FUNCTION_BLOCK Equipo_Valvula_5_2
VAR_INPUT
	PE 	  					  : BOOL;	//Parada de emergência
	Modo_Automatico           : BOOL;	//Modo automático
	Cmd_Auto         		  : BOOL;	//Comando automático
	Valv_Abierta		   	  : BOOL;	//Válvula aberta
	Valv_Cerrada			  : BOOL;	//Válvula fechada
	T_Discrepancia            : TIME;	//Tempo para erro de abertura
END_VAR
VAR_OUTPUT
	Activa_Equipo	 	      : BOOL;	//Aciona equipamento
	Estado					  : INT;	//Status da válvula
	Alr_Discrepancia		  : BOOL;	//Alarme de falha no acionamento
END_VAR
VAR_IN_OUT
	Cmd_Man 				  : BOOL;	//Comando manual
	Alarma				      : BOOL;	//Alarme
	Reset_Alarma		      : BOOL;	//Reset alarmes
END_VAR
VAR_STAT
	FP_Reset				  : R_TRIG;
	FN_Parada_Auto			  : F_TRIG;
	FP_Marcha_Auto            : R_TRIG;
	Cmd_Auto_interno		  :BOOL;	
END_VAR

VAR PERSISTENT
	Reset_Eventos         	  : BOOL;
	Timer_Discrepancia		  : TON;
	TON_TempoAbertura: TON;
	R_TRIG_TempoAbertura: R_TRIG;
	TempoAbertura	:DINT;	//Tempo que a válvula demora para abrir
	Eventos_Parciales		  : DINT;
	Eventos_Totales			  : DINT;
END_VAR
VAR // added by the converter: edge detectors and wires of the graphical bodies
    _w1, _w2, _w3, _w4, _w5, _w6, _w7 : BOOL;
    _rt1 : R_TRIG;
END_VAR

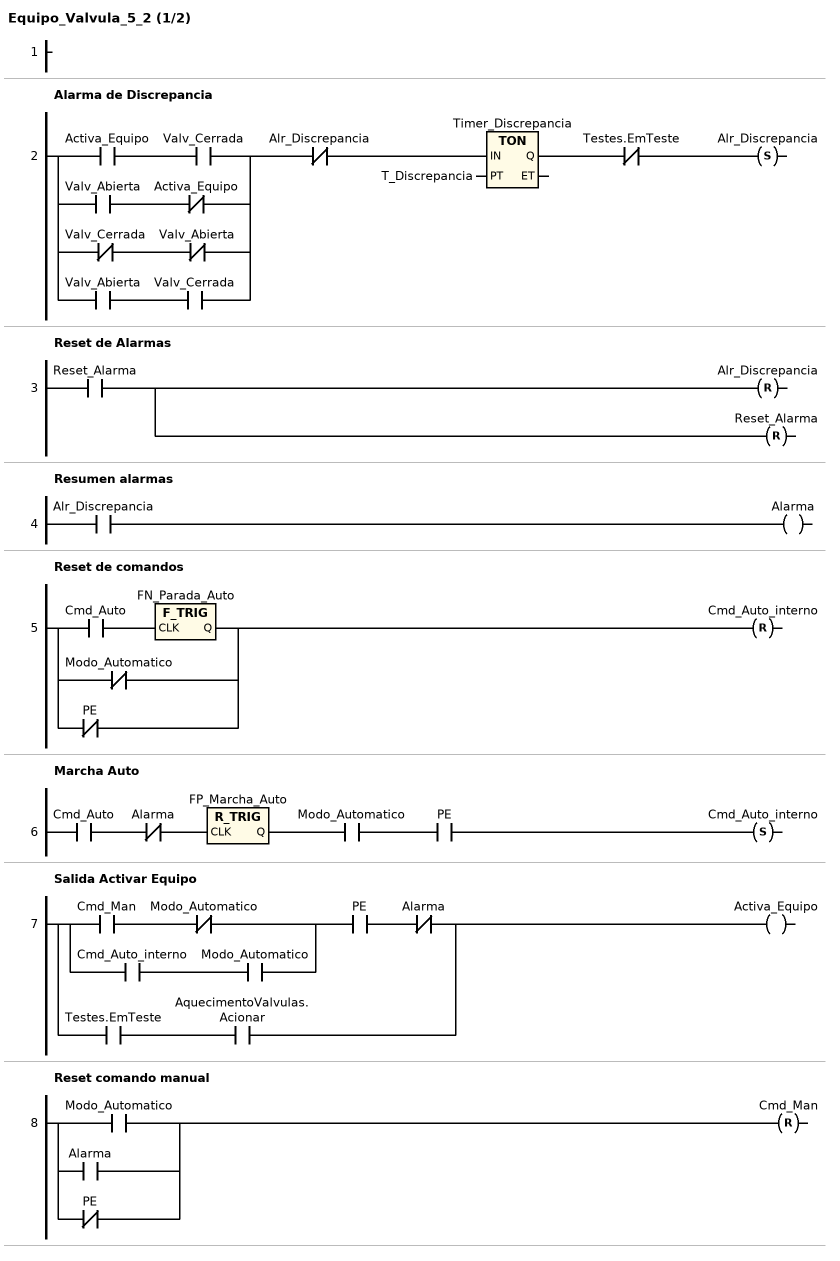
// NETWORK 1

// NETWORK 2: Alarma de Discrepancia
Timer_Discrepancia(IN := (Activa_Equipo AND Valv_Cerrada OR Valv_Abierta AND NOT Activa_Equipo OR NOT Valv_Cerrada AND NOT Valv_Abierta OR Valv_Abierta AND Valv_Cerrada) AND NOT Alr_Discrepancia, PT := T_Discrepancia); // TON
Alr_Discrepancia S= Timer_Discrepancia.Q AND NOT Testes.EmTeste;

// NETWORK 3: Reset de Alarmas
Alr_Discrepancia R= Reset_Alarma;
Reset_Alarma R= Reset_Alarma;

// NETWORK 4: Resumen alarmas
Alarma := Alr_Discrepancia;

// NETWORK 5: Reset de comandos
FN_Parada_Auto(CLK := Cmd_Auto); // F_TRIG
Cmd_Auto_interno R= FN_Parada_Auto.Q OR NOT Modo_Automatico OR NOT PE;

// NETWORK 6: Marcha Auto
FP_Marcha_Auto(CLK := Cmd_Auto AND NOT Alarma); // R_TRIG
Cmd_Auto_interno S= FP_Marcha_Auto.Q AND Modo_Automatico AND PE;

// NETWORK 7: Salida Activar Equipo
Activa_Equipo := (Cmd_Man AND NOT Modo_Automatico OR Cmd_Auto_interno AND Modo_Automatico) AND PE AND NOT Alarma OR Testes.EmTeste AND AquecimentoValvulas.Acionar;

// NETWORK 8: Reset comando manual
Cmd_Man R= Modo_Automatico OR Alarma OR NOT PE;

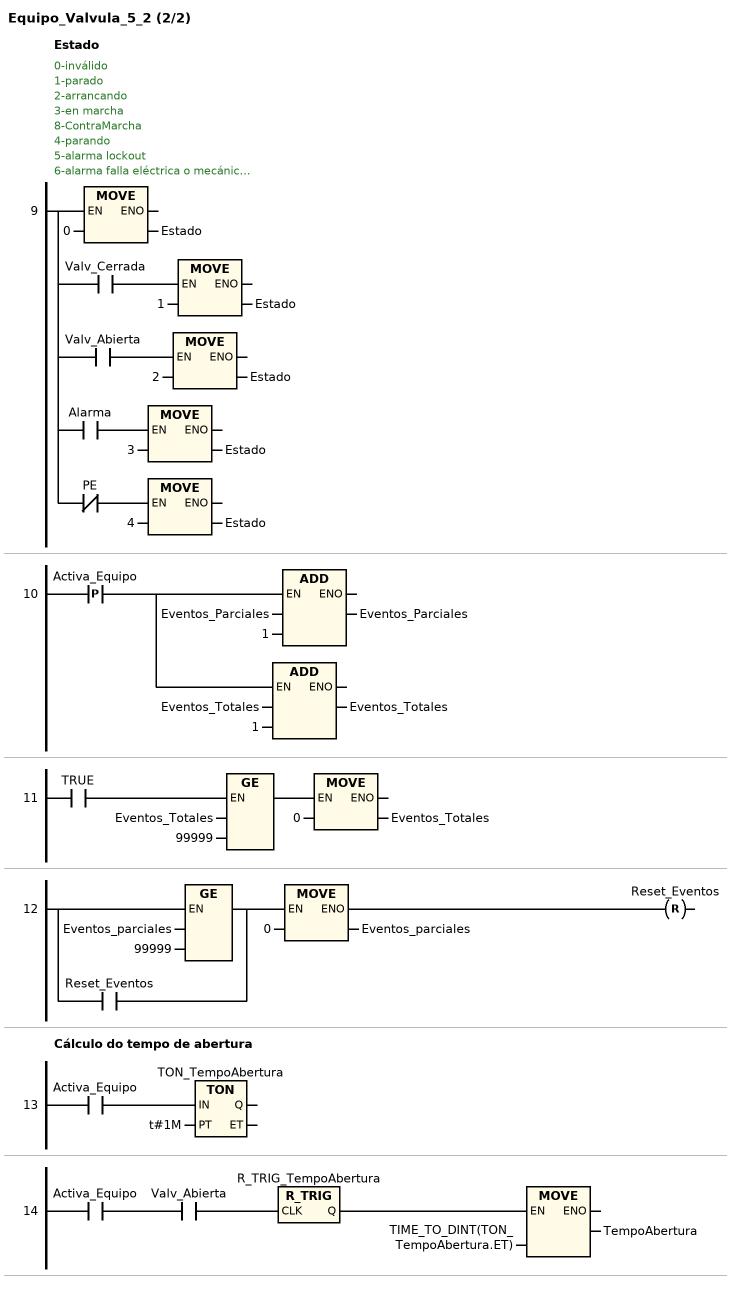
// NETWORK 9: Estado
// 0-inválido
// 1-parado
// 2-arrancando
// 3-en marcha
// 8-ContraMarcha
// 4-parando
// 5-alarma lockout
// 6-alarma falla eléctrica o mecánica
// 7-alarma pulsador emergencia
Estado := 0;
_w1 := Valv_Cerrada;
IF _w1 THEN Estado := 1; END_IF
_w2 := Valv_Abierta;
IF _w2 THEN Estado := 2; END_IF
_w3 := Alarma;
IF _w3 THEN Estado := 3; END_IF
_w4 := NOT PE;
IF _w4 THEN Estado := 4; END_IF

// NETWORK 10
_rt1(CLK := Activa_Equipo);
_w5 := _rt1.Q;
IF _w5 THEN Eventos_Parciales := Eventos_Parciales + 1; END_IF
_w6 := _rt1.Q;
IF _w6 THEN Eventos_Totales := Eventos_Totales + 1; END_IF

// NETWORK 11
IF Eventos_Totales >= 99999 THEN Eventos_Totales := 0; END_IF

// NETWORK 12
_w7 := Reset_Eventos;
IF NOT _w7 THEN
    _w7 := Eventos_parciales >= 99999;
END_IF
IF _w7 THEN Eventos_parciales := 0; END_IF
Reset_Eventos R= _w7;

// NETWORK 13: Cálculo do tempo de abertura
TON_TempoAbertura(IN := Activa_Equipo, PT := t#1M); // TON

// NETWORK 14
R_TRIG_TempoAbertura(CLK := Activa_Equipo AND Valv_Abierta); // R_TRIG
IF R_TRIG_TempoAbertura.Q THEN TempoAbertura := TIME_TO_DINT(TON_TempoAbertura.ET); END_IF

END_FUNCTION_BLOCK

(* stored: Version 1.1.0.1, ProductVersion 3.1.4024.14
   POU Equipo_Valvula_5_2: Id {06626da1-143b-442d-b3fe-2afb301794fa}, SpecialFunc None *)
